Fanuc KAREL source: port_WDO.kl

PROGRAM TP
%NOLOCKGROUP
VAR
 x: BOOLEAN
BEGIN
 x = WDO[3]
END TP
